{attribute 'GeneratedUsingTerminal: AT2050-5500-0018'}
{attribute addProperty BoxType "AT2050-5500-0018"}
{attribute addProperty Id "ControlAT %Q*UINT2"}
{attribute addProperty CRC "3674028256"}
{attribute addProperty Size "2"}
TYPE FB_Outputs_DAFD38E0 EXTENDS OutputBase_10CEE7DE :
STRUCT
	{attribute addProperty Name "Control"}
	Control AT %Q* : UINT;
END_STRUCT
END_TYPE

(* stored: Version 1.2.0.0, ProductVersion 3.1.4024.9
   DUT FB_Outputs_DAFD38E0: Id {f6a70c35-aed6-40fb-afe1-3c347694cad6} *)
